SYSTEM CrossingSubappConnectionCommandTest
  (* Version 1.0, 2022-06-29, AK115394 *)
  APPLICATION EventConnectionTestApp
    FBS
      fb_destinationevent : fb_destinationevent;
      fb_destinationevent_1 : fb_destinationevent;
      fb_destinationevent_2 : fb_sourceevent;
      fb_destinationevent_3 : fb_sourceevent;
      fb_destinationevent_4 : fb_sourceevent;
      fb_destinationevent_5 : fb_sourceevent;
      fb_destinationevent_6 : fb_sourceevent;
      fb_destinationevent_7 : fb_sourceevent;
    END_FBS
    SUBAPPLICATION Test1 (* connection between subapp borders *)
      EVENT_INPUT
        source;
      END_EVENT
      EVENT_OUTPUT
        EO1;
      END_EVENT
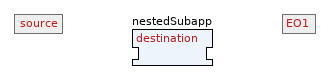
      SUBAPPLICATION nestedSubapp
        EVENT_INPUT
          destination;
        END_EVENT
      END_SUBAPPLICATION
    END_SUBAPPLICATION
    SUBAPPLICATION Test1Result
      EVENT_INPUT
        source;
      END_EVENT
      EVENT_OUTPUT
        EO1;
      END_EVENT
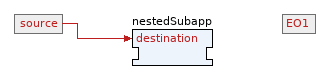
      SUBAPPLICATION nestedSubapp
        EVENT_INPUT
          destination;
        END_EVENT
      END_SUBAPPLICATION
      EVENT_CONNECTIONS
        source TO nestedSubapp.destination;
      END_CONNECTIONS
    END_SUBAPPLICATION
    SUBAPPLICATION Test2 (* connection between subapp borders, swap needed *)
      EVENT_INPUT
        destination;
      END_EVENT
      EVENT_OUTPUT
        EO1;
      END_EVENT
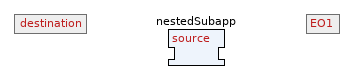
      SUBAPPLICATION nestedSubapp
        EVENT_INPUT
          source;
        END_EVENT
      END_SUBAPPLICATION
    END_SUBAPPLICATION
    SUBAPPLICATION Test2Solution
      EVENT_INPUT
        destination;
      END_EVENT
      EVENT_OUTPUT
        EO1;
      END_EVENT
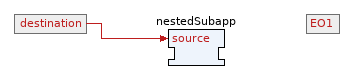
      SUBAPPLICATION nestedSubapp
        EVENT_INPUT
          source;
        END_EVENT
      END_SUBAPPLICATION
      EVENT_CONNECTIONS
        destination TO nestedSubapp.source;
      END_CONNECTIONS
    END_SUBAPPLICATION
    SUBAPPLICATION Test3Solution
      EVENT_INPUT
        destination;
      END_EVENT
      EVENT_OUTPUT
        EO1;
      END_EVENT
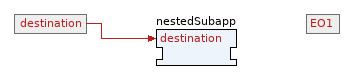
      SUBAPPLICATION nestedSubapp
        EVENT_INPUT
          destination;
        END_EVENT
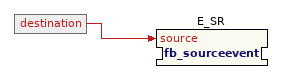
        FBS
          E_SR : fb_sourceevent;
        END_FBS
        EVENT_CONNECTIONS
          destination TO E_SR.source;
        END_CONNECTIONS
      END_SUBAPPLICATION
      EVENT_CONNECTIONS
        destination TO nestedSubapp.destination;
      END_CONNECTIONS
    END_SUBAPPLICATION
    SUBAPPLICATION Test3 (* crossing connection from FB to subapp border *)
      EVENT_INPUT
        destination;
      END_EVENT
      EVENT_OUTPUT
        EO1;
      END_EVENT
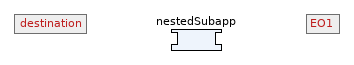
      SUBAPPLICATION nestedSubapp
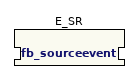
        FBS
          E_SR : fb_sourceevent;
        END_FBS
      END_SUBAPPLICATION
    END_SUBAPPLICATION
    SUBAPPLICATION Test4 (* crossing connection from FB in nested subapp to FB via app network *)
      EVENT_OUTPUT
        EO1;
      END_EVENT
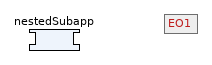
      SUBAPPLICATION nestedSubapp
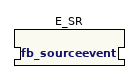
        FBS
          E_SR : fb_sourceevent;
        END_FBS
      END_SUBAPPLICATION
    END_SUBAPPLICATION
    SUBAPPLICATION Test4Solution
      EVENT_INPUT
        destination;
      END_EVENT
      EVENT_OUTPUT
        EO1;
      END_EVENT
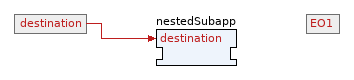
      SUBAPPLICATION nestedSubapp
        EVENT_INPUT
          destination;
        END_EVENT
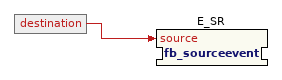
        FBS
          E_SR : fb_sourceevent;
        END_FBS
        EVENT_CONNECTIONS
          destination TO E_SR.source;
        END_CONNECTIONS
      END_SUBAPPLICATION
      EVENT_CONNECTIONS
        destination TO nestedSubapp.destination;
      END_CONNECTIONS
    END_SUBAPPLICATION
    SUBAPPLICATION Test5 (* crossing connection from FB to FB in nested subapp via app network *)
      EVENT_OUTPUT
        EO1;
      END_EVENT
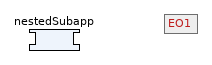
      SUBAPPLICATION nestedSubapp
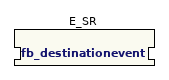
        FBS
          E_SR : fb_destinationevent;
        END_FBS
      END_SUBAPPLICATION
    END_SUBAPPLICATION
    SUBAPPLICATION Test5Solution
      EVENT_OUTPUT
        EO1;
        destination;
      END_EVENT
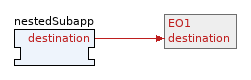
      SUBAPPLICATION nestedSubapp
        EVENT_OUTPUT
          destination;
        END_EVENT
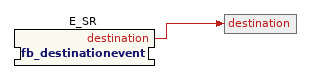
        FBS
          E_SR : fb_destinationevent;
        END_FBS
        EVENT_CONNECTIONS
          E_SR.destination TO destination;
        END_CONNECTIONS
      END_SUBAPPLICATION
      EVENT_CONNECTIONS
        nestedSubapp.destination TO destination;
      END_CONNECTIONS
    END_SUBAPPLICATION
    SUBAPPLICATION Test6 (* crossing connection from FB to nested subapp interface *)
      EVENT_OUTPUT
        EO1;
      END_EVENT
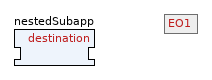
      SUBAPPLICATION nestedSubapp
        EVENT_OUTPUT
          destination;
        END_EVENT
      END_SUBAPPLICATION
    END_SUBAPPLICATION
    SUBAPPLICATION Test6Solution
      EVENT_OUTPUT
        EO1;
        destination;
      END_EVENT
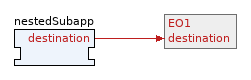
      SUBAPPLICATION nestedSubapp
        EVENT_OUTPUT
          destination;
        END_EVENT
      END_SUBAPPLICATION
      EVENT_CONNECTIONS
        nestedSubapp.destination TO destination;
      END_CONNECTIONS
    END_SUBAPPLICATION
    SUBAPPLICATION Test7 (* crossing connection from FB to FB in nested subapp, one pin already exists *)
      EVENT_OUTPUT
        destination;
      END_EVENT
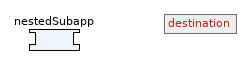
      SUBAPPLICATION nestedSubapp
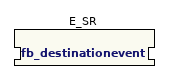
        FBS
          E_SR : fb_destinationevent;
        END_FBS
      END_SUBAPPLICATION
    END_SUBAPPLICATION
    SUBAPPLICATION Test7Solution
      EVENT_OUTPUT
        destination;
      END_EVENT
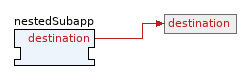
      SUBAPPLICATION nestedSubapp
        EVENT_OUTPUT
          destination;
        END_EVENT
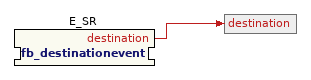
        FBS
          E_SR : fb_destinationevent;
        END_FBS
        EVENT_CONNECTIONS
          E_SR.destination TO destination;
        END_CONNECTIONS
      END_SUBAPPLICATION
      EVENT_CONNECTIONS
        nestedSubapp.destination TO destination;
      END_CONNECTIONS
    END_SUBAPPLICATION
    SUBAPPLICATION Test8 (* crossing connection from FB in subapp to FB in nested subapp *)
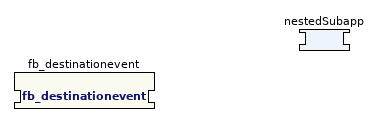
      FBS
        fb_destinationevent : fb_destinationevent;
      END_FBS
      SUBAPPLICATION nestedSubapp
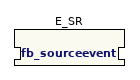
        FBS
          E_SR : fb_sourceevent;
        END_FBS
      END_SUBAPPLICATION
    END_SUBAPPLICATION
    SUBAPPLICATION Test8Solution
